// TIA Portal V18 export
FUNCTION "Regenaration program sequences" : Void   // FC23, LAD
{ S7_Optimized_Access := 'TRUE' }
VERSION : 0.1
// stored: AutoNumber true, IsIECCheckEnabled false, SetENOAutomatically false, UDAEnableTagReadback false
   VAR_TEMP
      temp1 : Bool;
   END_VAR
   VAR_TEMP   // added for the SCL form of the ladder/FBD networks
      _w1 : Bool;
   END_VAR
BEGIN

REGION Network 1: Function regeneration
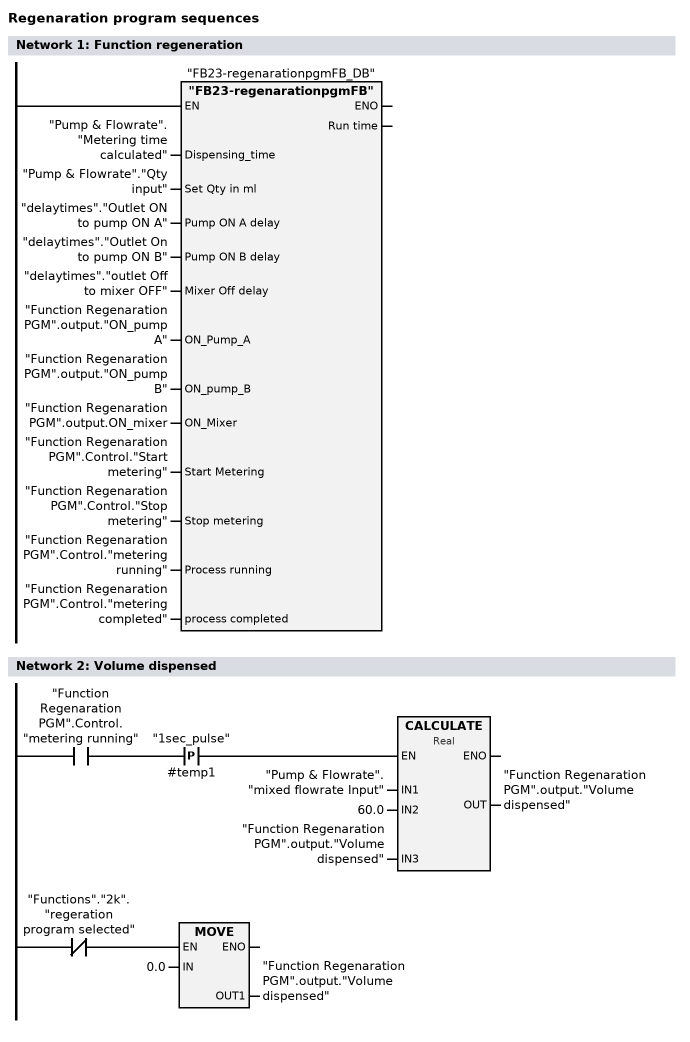
   RUNG wire#powerrail
      "FB23-regenarationpgmFB_DB"(Dispensing_time := "Pump & Flowrate"."Metering time calculated", "Set Qty in ml" := "Pump & Flowrate"."Qty input", "Pump ON A delay" := "delaytimes"."Outlet ON to pump ON A", "Pump ON B delay" := "delaytimes"."Outlet On to pump ON B", "Mixer Off delay" := "delaytimes"."outlet Off to mixer OFF", ON_Pump_A := "Function Regenaration PGM".output."ON_pump A", ON_pump_B := "Function Regenaration PGM".output."ON_pump B", ON_Mixer := "Function Regenaration PGM".output.ON_mixer, "Start Metering" := "Function Regenaration PGM".Control."Start metering", "Stop metering" := "Function Regenaration PGM".Control."Stop metering", "Process running" := "Function Regenaration PGM".Control."metering running", "process completed" := "Function Regenaration PGM".Control."metering completed", "Run time" =>)
   END_RUNG
   // the same network as SCL:
   "FB23-regenarationpgmFB_DB"(Dispensing_time := "Pump & Flowrate"."Metering time calculated",   // "FB23-regenarationpgmFB"
                           "Set Qty in ml" := "Pump & Flowrate"."Qty input",
                           "Pump ON A delay" := "delaytimes"."Outlet ON to pump ON A",
                           "Pump ON B delay" := "delaytimes"."Outlet On to pump ON B",
                           "Mixer Off delay" := "delaytimes"."outlet Off to mixer OFF",
                           ON_Pump_A := "Function Regenaration PGM".output."ON_pump A",
                           ON_pump_B := "Function Regenaration PGM".output."ON_pump B",
                           ON_Mixer := "Function Regenaration PGM".output.ON_mixer,
                           "Start Metering" := "Function Regenaration PGM".Control."Start metering",
                           "Stop metering" := "Function Regenaration PGM".Control."Stop metering",
                           "Process running" := "Function Regenaration PGM".Control."metering running",
                           "process completed" := "Function Regenaration PGM".Control."metering completed");
END_REGION

REGION Network 2: Volume dispensed
   RUNG wire#powerrail
      Contact( "Function Regenaration PGM".Control."metering running" )
      P_Contact(operand := "1sec_pulse", bit := #temp1)
      { S7_Templates := "SrcType := Real"; S7_Expression := "(IN1/IN2)+IN3" } Calculate(in1 := "Pump & Flowrate"."mixed flowrate Input", in2 := 60.0, in3 := "Function Regenaration PGM".output."Volume dispensed", out => "Function Regenaration PGM".output."Volume dispensed")
   END_RUNG
   RUNG wire#powerrail
      I_Contact( "Functions"."2k"."regeration program selected" )
      Move(in := 0.0, out1 => "Function Regenaration PGM".output."Volume dispensed")
   END_RUNG
   // the same network as SCL:
   #_w1 := "Function Regenaration PGM".Control."metering running" AND "1sec_pulse" AND NOT #temp1;   // rising edge of "1sec_pulse"
   #temp1 := "1sec_pulse";
   IF #_w1 THEN
       "Function Regenaration PGM".output."Volume dispensed" := ("Pump & Flowrate"."mixed flowrate Input"/60.0)+"Function Regenaration PGM".output."Volume dispensed";
   END_IF;
   IF NOT "Functions"."2k"."regeration program selected" THEN
       "Function Regenaration PGM".output."Volume dispensed" := 0.0;
   END_IF;
END_REGION
END_FUNCTION
